ABB RobotStudio station: Projekt_2__159557_161672 (1).rspag

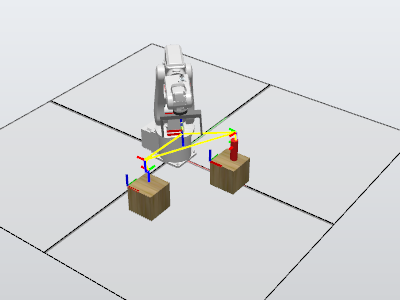
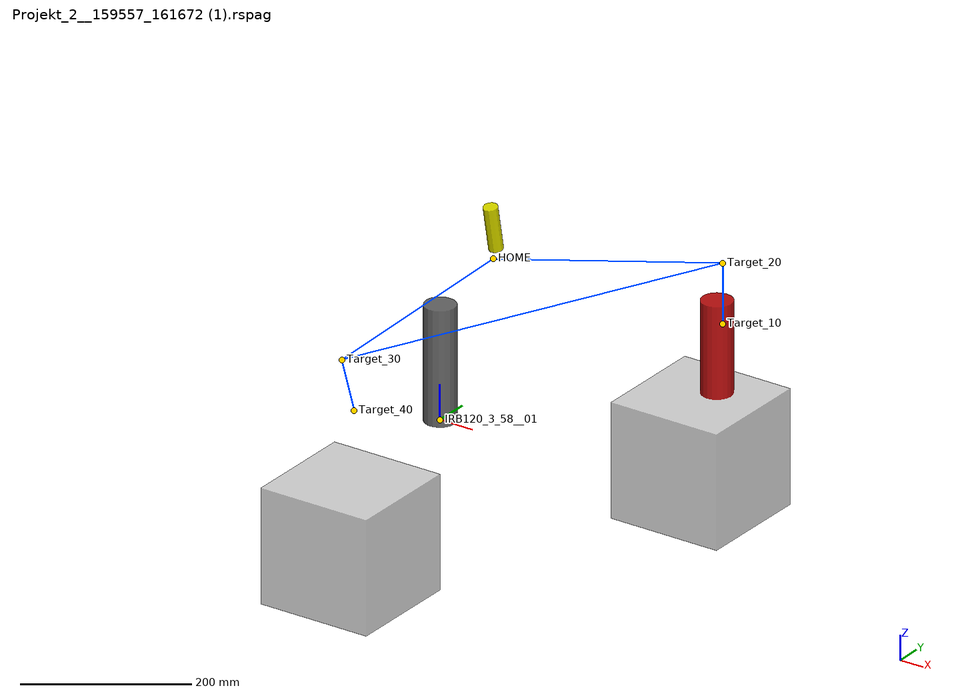
[picture v1: parts stored in the station drawn from their meshes, with robot base, taught points and paths (robot models come from the ABB library and are not in the file)]
--- station ---
Station grip (saved by RobotStudio 25.5.11605.0)
Controller Controller3
  mechanical unit ROB_1: IRB120_3_58__01, 6 joints, base frame (0, 0, 0) mm
Layout (positions relative to the parent item):
  - TOOL1 [mechanism] at (251.76, -263.69, 503.18) mm, rotated rx 179.45 ry 3.37 rz -141.19 deg; joint values [0, 0] (rad or m)
      TCP TOOL1_1 at (100, 20, 100) mm
      TCP TOOL1_2 at (100, 20, 120) mm
      links: BAZA, L1, L2
  - SmartComponent_1 [smart component]
      signals: DI OTW_CHWYTAK, DI ZAMKNIJ_CHWYTAK, DO chwycil, DO puscil
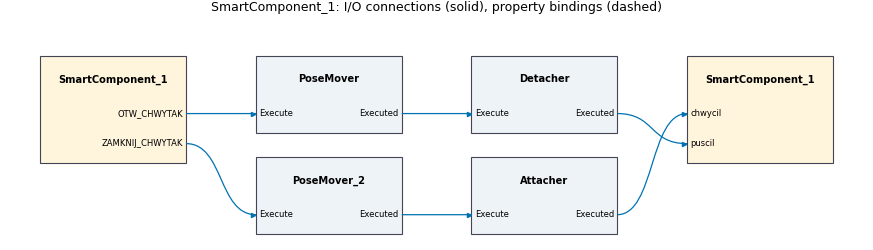
      connections:
        SmartComponent_1.OTW_CHWYTAK -> PoseMover.Execute
        SmartComponent_1.ZAMKNIJ_CHWYTAK -> PoseMover_2.Execute
        PoseMover_2.Executed -> Attacher.Execute
        PoseMover.Executed -> Detacher.Execute
        Attacher.Executed -> SmartComponent_1.chwycil
        Detacher.Executed -> SmartComponent_1.puscil
    - PoseMover [smart component, from Components\PoseMover.rslib]
        properties: Mechanism=TOOL1; Pose=1; Duration=0
    - PoseMover_2 [smart component, from Components\PoseMover.rslib]
        properties: Mechanism=TOOL1; Pose=2; Duration=0
    - Attacher [smart component, from Components\Attacher.rslib]
        properties: Parent=TOOL1; Flange=0; Child=OBIEKT; Mount=false; Offset=[0 0 0]; Orientation=[0 0 0]
    - Detacher [smart component, from Components\Detacher.rslib]
        properties: Child=OBIEKT; KeepPosition=true
  - IRB120_3_58__01 [mechanism, from %ABB.RobotStudio.Models.IRB120%\IRB120_3_58_G_01.rslib] at (0, 0, 0) mm; joint values [-0.8203, 0.2075, -0.047, 0.0602, 1.4159, -1.5073] (rad or m)
  - LineSensor [smart component, from Components\LineSensor.rslib] at (254.32, -261.48, 452.59) mm, rotated rx 174.08 ry 5.49 rz -149.06 deg
      properties: Start=[-2.68170960104896E-06 7.89233661852608E-05 0.000996850385733661]; End=[-0.000454564178909378 0.00295577462179693 0.0597642894833072]; Length=0.0588395476614156; Radius=0.00914634146341463; Tag=(none); SenseMultiple=false; SensedPart=OBIEKT; SensedPoint=[0.195780838012695 -0.444558288574219 0.274601440429687]
    - _sensorPart_ [part], size 18.5 x 20.9 x 59.7 mm
  - Part_7 [part], size 40 x 39.4 x 150 mm
  - OBIEKT [part] at (401.12, -10.76, 151.92) mm, size 40 x 40 x 120 mm
  - STOLIK1 [part] at (312.5, -99.53, 0) mm, size 150 x 150 x 150 mm
  - STOLIK2 [part] at (108.95, -519.83, 0) mm, size 150 x 150 x 150 mm
Attachment: TOOL1 is attached to IRB120_3_58__01 / Link6
Attachment: LineSensor is attached to TOOL1 / BAZA
Attachment: STOLIK1_WOBJ is attached to STOLIK1
Attachment: STOLIK2_WOBJ is attached to STOLIK2
Station signals: DI MAN_OT, DI MAN_ZAM
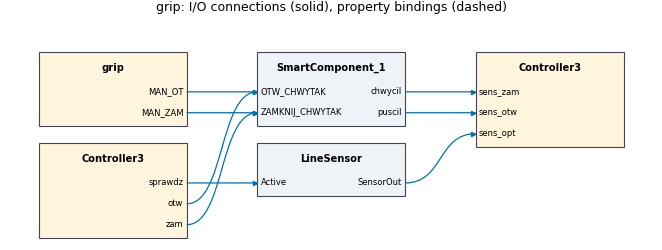
Station logic (signal -> signal, property => property):
  grip.MAN_OT -> SmartComponent_1.OTW_CHWYTAK
  grip.MAN_ZAM -> SmartComponent_1.ZAMKNIJ_CHWYTAK
  SmartComponent_1.chwycil -> Controller3.sens_zam
  SmartComponent_1.puscil -> Controller3.sens_otw
  LineSensor.SensorOut -> Controller3.sens_opt
  Controller3.sprawdz -> LineSensor.Active
  Controller3.otw -> SmartComponent_1.OTW_CHWYTAK
  Controller3.zam -> SmartComponent_1.ZAMKNIJ_CHWYTAK

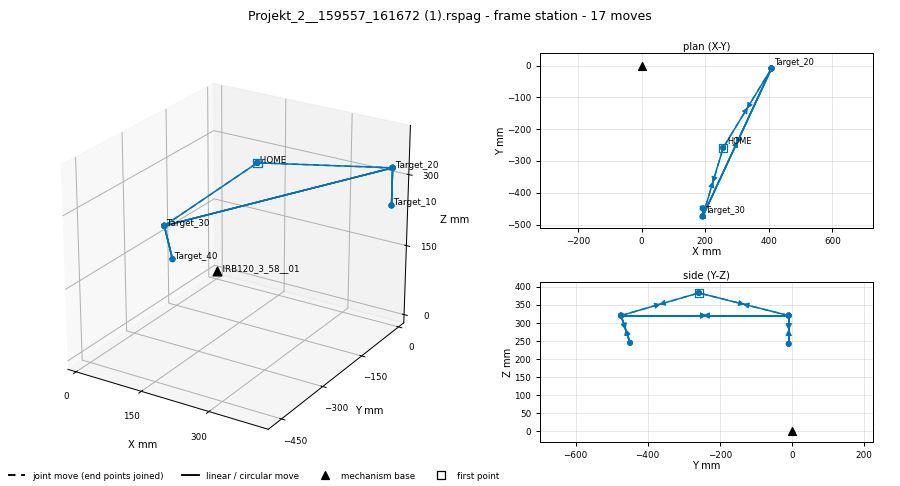
[picture p0: tool path of Projekt_2__159557_161672 (1).rspag in frame station, 17 of 17 moves have a stored position in this frame; points joined in program order, loops and branches not executed]
--- Backups/Controller3/RAPID/TASK1/PROGMOD/CalibData.mod ---
MODULE CalibData
    PERS tooldata TOOL1_1:=[TRUE,[[0,0,100],[1,0,0,0]],[1,[0,0,50],[1,0,0,0],0,0,0]];
    PERS tooldata TOOL1_2:=[TRUE,[[0,0,120],[1,0,0,0]],[1,[0,0,50],[1,0,0,0],0,0,0]];
    TASK PERS wobjdata STOLIK1_WOBJ:=[FALSE,TRUE,"",[[312.5,-99.532,150],[1,0,0,0]],[[0,0,0],[1,0,0,0]]];
    TASK PERS wobjdata STOLIK2_WOBJ:=[FALSE,TRUE,"",[[108.946,-517.788,150],[1,0,0,0]],[[0,0,0],[1,0,0,0]]];
ENDMODULE

--- Backups/Controller3/RAPID/TASK1/PROGMOD/Module1.mod ---
MODULE Module1
    CONST robtarget HOME:=[[256.540799784,-258.359619211,383.3890458],[0.026170031,-0.332202085,0.942736232,0.014328322],[-1,0,-1,0],[9E+09,9E+09,9E+09,9E+09,9E+09,9E+09]];
    CONST robtarget Target_20:=[[95.936093413,90.500324625,170.655659821],[0.019267747,-0.648961154,0.760236312,0.022779921],[-1,0,-1,0],[9E+09,9E+09,9E+09,9E+09,9E+09,9E+09]];
    CONST robtarget Target_10:=[[95.936098518,90.500325424,92.212250372],[0.019267765,-0.64896114,0.760236324,0.022779908],[-1,0,-1,0],[9E+09,9E+09,9E+09,9E+09,9E+09,9E+09]];
    CONST robtarget Target_30:=[[83.318009304,43.822023982,170.655580274],[0.029537862,0.02069217,0.999340613,0.004205714],[-1,0,-1,0],[9E+09,9E+09,9E+09,9E+09,9E+09,9E+09]];
    CONST robtarget Target_40:=[[83.317976738,68.822032986,95.066160203],[0.006133318,-0.020829065,-0.999758234,-0.003464862],[-1,-1,-1,0],[9E+09,9E+09,9E+09,9E+09,9E+09,9E+09]];
    !***********************************************************
    !
    ! Module:  Module1
    !
    ! Description:
    !   <Insert description here>
    !
    ! Author: Kamil
    !
    ! Version: 1.0
    !
    !***********************************************************


    !***********************************************************
    !
    ! Procedure main
    !
    !   This is the entry point of your program
    !
    !***********************************************************
    PROC main()
        Path_10;
    ENDPROC
    PROC Path_10()
        Reset sprawdz;
        Reset zam;
        Set otw;
        WaitTime 0.5;
        Reset otw;

        WHILE TRUE DO
            MoveJ HOME, v100, fine, TOOL1_2\WObj:=wobj0;
            MoveL Target_20, v100, z50, TOOL1_2\WObj:=STOLIK1_WOBJ;
            MoveL Target_10, v100, fine, TOOL1_2\WObj:=STOLIK1_WOBJ;

            Set sprawdz;
            WaitTime 0.2;

            IF TestDI(sens_opt) THEN
                Set zam;
                WaitTime 0.5;
                Reset zam;
                Reset sprawdz;
                MoveL Target_20, v100, z50, TOOL1_2\WObj:=STOLIK1_WOBJ;
                MoveL Target_30, v100, z50, TOOL1_2\WObj:=STOLIK2_WOBJ;
                MoveL Target_40, v100, fine, TOOL1_2\WObj:=STOLIK2_WOBJ;

                Set otw;
                WaitTime 0.5;
                Reset otw;

                MoveL Target_30, v100, z50, TOOL1_2\WObj:=STOLIK2_WOBJ;
            ELSE
                Reset sprawdz;
                MoveL Target_20, v100, z50, TOOL1_2\WObj:=STOLIK1_WOBJ;
                MoveJ HOME, v100, fine, TOOL1_2\WObj:=wobj0;

                MoveL Target_30, v100, z50, TOOL1_2\WObj:=STOLIK2_WOBJ;
                MoveL Target_40, v100, fine, TOOL1_2\WObj:=STOLIK2_WOBJ;

                Set sprawdz;
                WaitTime 0.2;

                IF TestDI(sens_opt) THEN
                    Set zam;
                    WaitTime 0.5;
                    Reset zam;
                    Reset sprawdz;

                    MoveL Target_30, v100, z50, TOOL1_2\WObj:=STOLIK2_WOBJ;
                    MoveL Target_20, v100, z50, TOOL1_2\WObj:=STOLIK1_WOBJ;
                    MoveL Target_10, v100, fine, TOOL1_2\WObj:=STOLIK1_WOBJ;

                    Set otw;
                    WaitTime 0.5;
                    Reset otw;

                    MoveL Target_20, v100, z50, TOOL1_2\WObj:=STOLIK1_WOBJ;
                ELSE
                    Reset sprawdz;
                    MoveL Target_30, v100, z50, TOOL1_2\WObj:=STOLIK2_WOBJ;
                ENDIF
            ENDIF
            MoveJ HOME, v100, fine, TOOL1_2\WObj:=wobj0;
        ENDWHILE
    ENDPROC
ENDMODULE

--- Backups/Controller3/SYSPAR/EIO.cfg ---
EIO:CFG_1.0:6:1::
#
EIO_SIGNAL:

      -Name "syg2" -SignalType "DO"

      -Name "otw" -SignalType "DO"

      -Name "zam" -SignalType "DO"

      -Name "sens_opt" -SignalType "DI"

      -Name "sens_otw" -SignalType "DI"

      -Name "sens_zam" -SignalType "DI"

      -Name "sprawdz" -SignalType "DO"
